// TIA Portal V20 export
TYPE "LConSMC_typeDiamCalcDiag"
// Diagnosestruktur des Durchmesserrechners / Diagnostic strukture of diameter calculation
// stored: Access Published
   STRUCT
      atMinDia : Bool := FALSE;   // TRUE: Minimaler Durchmesser erreicht / TRUE: Diameter calculation has reached minimum diameter
      atMaxDia : Bool := FALSE;   // TRUE: Maximaler Durchmesser erreicht / TRUE: Diameter calculation has reached maximum diameter
      diamIsHold : Bool := FALSE;   // TRUE: Durchmesserrechner ist gestoppt: - Bahngeschwindigkeit < diamConfig.minLineVelo - Wicklerdrehzahl < diamConfig.minShaftSpeed - Eingang "holdDiameter" = TRUE / TRUE: Diameter calculation is hold: line velocity < diamConfig.minLineVelo shaftSpeed < diamConfig.minShaftSpeed input "holdDiameter" = TRUE
      calculatedWebThickness : LReal;   // Berechnete Materialdicke Nur relevant in den Modi Integral (2) und Position (5) / Calculated web thickness Only relevant for calculation modes integral (2) and position (5)
   END_STRUCT;
END_TYPE
